Omron CX-Programmer project NewProject (CX-Programmer 9.61)

# PLC NewPLC1: CP1H XA

## Global symbols (name address type ; comment)
0.00 BOOL  ; start
0.01 BOOL  ; Dsens1
0.02 BOOL  ; Dsens2
0.03 BOOL  ; Detector
0.05 BOOL  ; stop
100.00 BOOL  ; Convayer
100.01 BOOL  ; Roller_stop
100.02 BOOL  ; Convayer1
100.03 BOOL  ; Place1_z
100.04 BOOL  ; Place1_Grab
100.05 BOOL  ; Place1_x
100.06 BOOL  ; Convayer2
10.00 BOOL  ; M1
10.01 BOOL  ; M2
10.02 BOOL  ; M3
10.03 BOOL  ; M4
10.04 BOOL  ; M5
1.00 BOOL  ; Mstart
1.01 BOOL  ; Mstop
T0000 BOOL  ; Timer1
T0001 BOOL  ; Timer2
T0002 BOOL  ; Timer3
T0003 BOOL  ; Timer4
T0004 BOOL  ; Timer5
T0005 BOOL  ; Timer6
T0006 BOOL  ; Timer7
T0007 BOOL  ; Timer8
T0008 BOOL  ; Timer9

## Program NewProgram1 (cyclic task 0)

### Section Section1

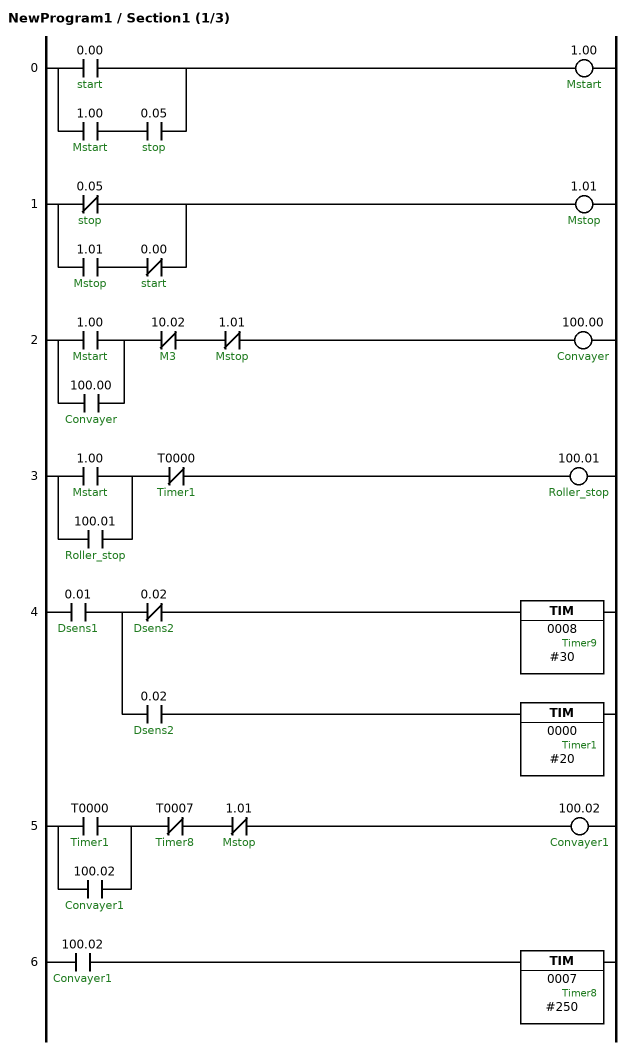
; rung 0
LD 0.00  ; start
LD 1.00  ; Mstart
AND 0.05  ; stop
ORLD
OUT 1.00  ; Mstart
; rung 1
LDNOT 0.05  ; stop
LD 1.01  ; Mstop
ANDNOT 0.00  ; start
ORLD
OUT 1.01  ; Mstop
; rung 2
LD 1.00  ; Mstart
OR 100.00  ; Convayer
ANDNOT 10.02  ; M3
ANDNOT 1.01  ; Mstop
OUT 100.00  ; Convayer
; rung 3
LD 1.00  ; Mstart
OR 100.01  ; Roller_stop
ANDNOT T0000  ; Timer1
OUT 100.01  ; Roller_stop
; rung 4
LD 0.01  ; Dsens1
OUT TR0
ANDNOT 0.02  ; Dsens2
TIM 0008 #30  ; Timer9
LD TR0
AND 0.02  ; Dsens2
TIM 0000 #20  ; Timer1
; rung 5
LD T0000  ; Timer1
OR 100.02  ; Convayer1
ANDNOT T0007  ; Timer8
ANDNOT 1.01  ; Mstop
OUT 100.02  ; Convayer1
; rung 6
LD 100.02  ; Convayer1
TIM 0007 #250  ; Timer8

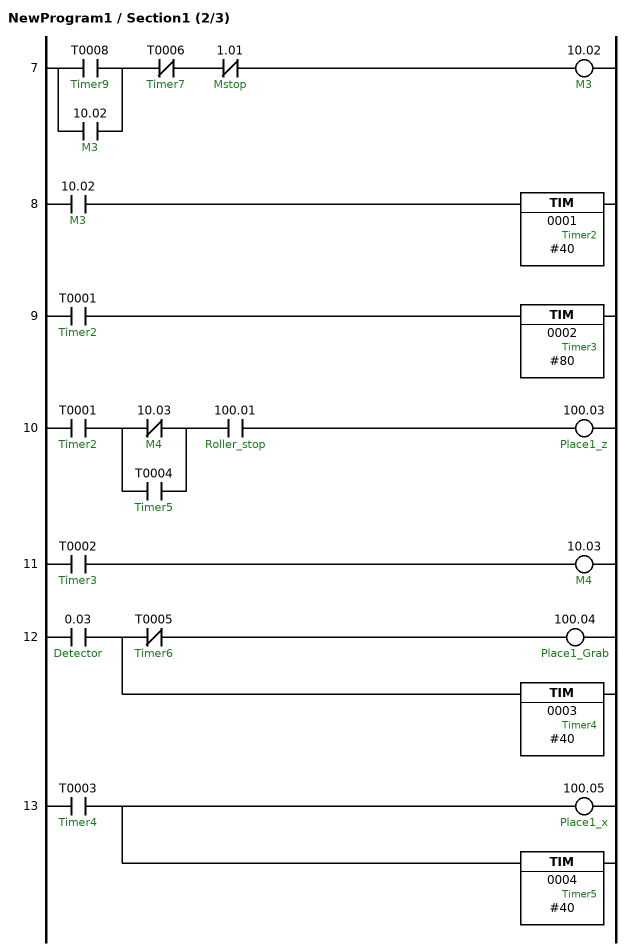
; rung 7
LD T0008  ; Timer9
OR 10.02  ; M3
ANDNOT T0006  ; Timer7
ANDNOT 1.01  ; Mstop
OUT 10.02  ; M3
; rung 8
LD 10.02  ; M3
TIM 0001 #40  ; Timer2
; rung 9
LD T0001  ; Timer2
TIM 0002 #80  ; Timer3
; rung 10
LD T0001  ; Timer2
LDNOT 10.03  ; M4
OR T0004  ; Timer5
ANDLD
AND 100.01  ; Roller_stop
OUT 100.03  ; Place1_z
; rung 11
LD T0002  ; Timer3
OUT 10.03  ; M4
; rung 12
LD 0.03  ; Detector
OUT TR0
ANDNOT T0005  ; Timer6
OUT 100.04  ; Place1_Grab
LD TR0
TIM 0003 #40  ; Timer4
; rung 13
LD T0003  ; Timer4
OUT 100.05  ; Place1_x
TIM 0004 #40  ; Timer5

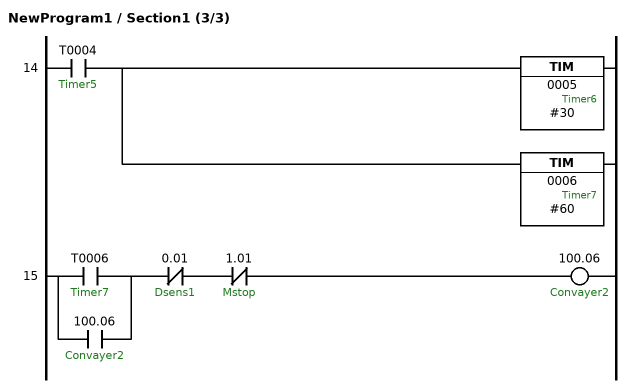
; rung 14
LD T0004  ; Timer5
TIM 0005 #30  ; Timer6
TIM 0006 #60  ; Timer7
; rung 15
LD T0006  ; Timer7
OR 100.06  ; Convayer2
ANDNOT 0.01  ; Dsens1
ANDNOT 1.01  ; Mstop
OUT 100.06  ; Convayer2

### Section END
; rung 0
END(001)